FUNCTION_BLOCK FINAL FB_PackML
VAR_IN_OUT
	PackML							: ST_PMLData;
	Control							: ST_System;
END_VAR
VAR
	_Cfg_ModeTransitions			: ARRAY[0..9, 0..31] OF BOOL;
	_Index							: INT;
	_LastState						: DINT;
	_LastUnit						: DINT;
	_MessageClearPointer			: INT;
	_WarningRefreshPointer			: INT;
	_WarningRefresh					: F_TRIG;
END_VAR
VAR CONSTANT
	_MaxModeLength					: INT := 7;
	_MaxStateLength					: INT := 17;
END_VAR
VAR PERSISTENT
	_LS_H_IndicatorMatrix				: ARRAY[0..31] OF DINT :=[1032,33792,1032,361504,66784,361504,198690,67616,1028,1028,1032,99360,1216,82984,295936,1032,1028];
	_PB_IndicatorMatrix					: ARRAY[0..31] OF DINT :=[0,256,32768,0,32768,32768,32768,16384,0,256,0,0,32768,32768,16384,32768,256,0];			
	_LS_H_IndicatorDescription			: ARRAY[0..31] OF STRING(40) := ['','Alarm','Abnormal Stop','Controlled Stop','','Alert','Starved Upstream','Blocked Downstream','','','Low Material','Material Exhausted','','','Alert','Alarm','Starting / Restarting','','','','','','','','','','','','',''];		
	_PB_IndicatorDescription			: ARRAY[0..31] OF STRING(40) := ['','','','','','','','','Ready to Reset','','','','','','Ready to Start','Running','','','','','','','','','','','','','','','',''];		
END_VAR

M_Administration();
M_Commands();
M_Indicators();
M_ModeControl();
M_SafetyBreach();
M_StateMapping();
M_StateTransitions();
M_TransitionCounts();

METHOD PRIVATE M_Administration
VAR_INPUT
END_VAR
VAR_INST
	_index					: INT;
END_VAR
IF PackML.Status.UnitModeCurrent > _maxModeLength THEN
	PackML.Control.UnitMode := 0;
	PackML.Status.UnitModeCurrent := 0;
END_IF

//Time spent in Mode
//The elapsed time the machine has spent in that mode since it entered that mode.  Array index is equal to designation of the mode.
IF PackML.Status.UnitModeChangeInProcess THEN
	PackML.Admin.ModeCurrentTime[PackML.Status.UnitModeCurrent] := 0;
END_IF
IF Control.SystemTime.SecondPulse THEN
	PackML.Admin.ModeCurrentTime[PackML.Status.UnitModeCurrent] := PackML.Admin.ModeCurrentTime[PackML.Status.UnitModeCurrent] + 1;
	IF PackML.Admin.ModeCurrentTime[PackML.Status.UnitModeCurrent] < 0 THEN
		PackML.Admin.ModeCurrentTime[PackML.Status.UnitModeCurrent] := 0;
	END_IF
	IF PackML.Admin.ResetTimerCounters THEN
		FOR _index := 0 TO _maxModeLength DO
			PackML.Admin.ModeCurrentTime[_index] := 0;
		END_FOR
	END_IF
END_IF

//Cumulative TIME In Each Mode
//The cumulative elapsed time the machine has spent in each mode since it’s timers and counters were reset.  
IF Control.SystemTime.SecondPulse THEN
	PackML.Admin.ModeCummulativeTime[PackML.Status.UnitModeCurrent] := PackML.Admin.ModeCummulativeTime[PackML.Status.UnitModeCurrent] + 1;
	IF PackML.Admin.ModeCummulativeTime[PackML.Status.UnitModeCurrent] < 0 THEN
		PackML.Admin.ModeCummulativeTime[PackML.Status.UnitModeCurrent] := 0;
	END_IF
	IF PackML.Admin.ResetTimerCounters THEN
		FOR _index := 0 TO _maxModeLength DO
			PackML.Admin.ModeCummulativeTime[_index] := 0;
		END_FOR
	END_IF
END_IF

//TIME spent in State
//The elapsed time the machine has spent in that State since it entered that State.  Array index is equal to designation of the mode.
IF PackML.Status.StateChangeInProgress THEN
	PackML.Admin.StateCurrentTime[PackML.Status.UnitModeCurrent,PackML.Status.StateCurrent] := 0;
END_IF
IF Control.SystemTime.SecondPulse THEN
	PackML.Admin.StateCurrentTime[PackML.Status.UnitModeCurrent,PackML.Status.StateCurrent] := PackML.Admin.StateCurrentTime[PackML.Status.UnitModeCurrent,PackML.Status.StateCurrent] + 1;
	IF PackML.Admin.StateCurrentTime[PackML.Status.UnitModeCurrent,PackML.Status.StateCurrent] < 0 THEN
		PackML.Admin.StateCurrentTime[PackML.Status.UnitModeCurrent,PackML.Status.StateCurrent] := 0;
	END_IF
	IF PackML.Admin.ResetTimerCounters THEN
		FOR _index := 0 TO _maxStateLength DO
			PackML.Admin.StateCurrentTime[PackML.Status.UnitModeCurrent,_index] := 0;
		END_FOR
	END_IF
END_IF

//Cumulative Time In Each Mode
//The cumulative elapsed time the machine has spent in each mode since it’s timers and counters were reset.  
IF Control.SystemTime.SecondPulse THEN
	PackML.Admin.StateCummulativeTime[PackML.Status.UnitModeCurrent,PackML.Status.StateCurrent] := PackML.Admin.StateCummulativeTime[PackML.Status.UnitModeCurrent,PackML.Status.StateCurrent] + 1;
	IF PackML.Admin.StateCummulativeTime[PackML.Status.UnitModeCurrent,PackML.Status.StateCurrent] < 0 THEN
		PackML.Admin.StateCummulativeTime[PackML.Status.UnitModeCurrent,PackML.Status.StateCurrent] := 0;
	END_IF
	IF PackML.Admin.ResetTimerCounters THEN
		FOR _index := 0 TO _maxStateLength DO
			PackML.Admin.StateCummulativeTime[PackML.Status.UnitModeCurrent,_index] := 0;
		END_FOR
	END_IF
END_IF
END_METHOD

METHOD PRIVATE M_Commands
VAR_INPUT
END_VAR
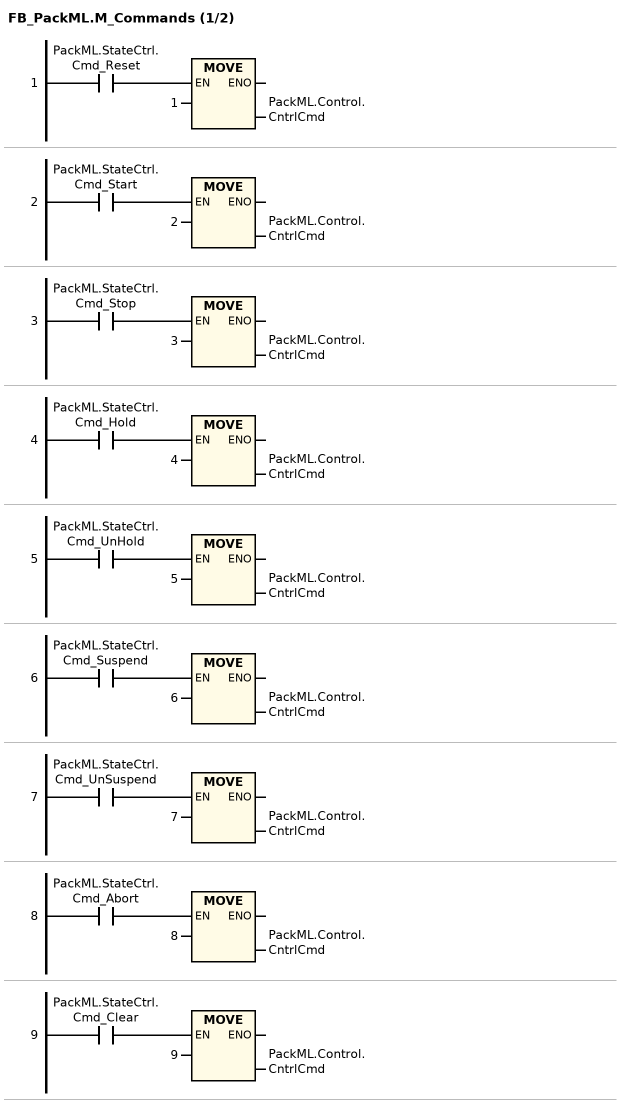
// NETWORK 1
IF PackML.StateCtrl.Cmd_Reset THEN PackML.Control.CntrlCmd := 1; END_IF

// NETWORK 2
IF PackML.StateCtrl.Cmd_Start THEN PackML.Control.CntrlCmd := 2; END_IF

// NETWORK 3
IF PackML.StateCtrl.Cmd_Stop THEN PackML.Control.CntrlCmd := 3; END_IF

// NETWORK 4
IF PackML.StateCtrl.Cmd_Hold THEN PackML.Control.CntrlCmd := 4; END_IF

// NETWORK 5
IF PackML.StateCtrl.Cmd_UnHold THEN PackML.Control.CntrlCmd := 5; END_IF

// NETWORK 6
IF PackML.StateCtrl.Cmd_Suspend THEN PackML.Control.CntrlCmd := 6; END_IF

// NETWORK 7
IF PackML.StateCtrl.Cmd_UnSuspend THEN PackML.Control.CntrlCmd := 7; END_IF

// NETWORK 8
IF PackML.StateCtrl.Cmd_Abort THEN PackML.Control.CntrlCmd := 8; END_IF

// NETWORK 9
IF PackML.StateCtrl.Cmd_Clear THEN PackML.Control.CntrlCmd := 9; END_IF

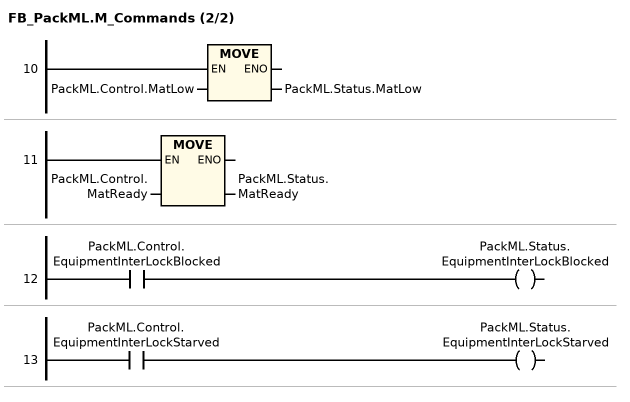
// NETWORK 10
PackML.Status.MatLow := PackML.Control.MatLow;

// NETWORK 11
PackML.Status.MatReady := PackML.Control.MatReady;

// NETWORK 12
PackML.Status.EquipmentInterLockBlocked := PackML.Control.EquipmentInterLockBlocked;

// NETWORK 13
PackML.Status.EquipmentInterLockStarved := PackML.Control.EquipmentInterLockStarved;
END_METHOD

METHOD PRIVATE M_Indicators
VAR_INST
	_i 		: DINT;
	_f_trig	: F_TRIG;
	_r_trig	: R_TRIG;
	k : bool;
END_VAR
PackML.Indicator.LS_H_Output := _LS_H_IndicatorMatrix[PackML.Status.StateCurrent];

//Red Lamp
IF PackML.Indicator.LS_H_Output.0 THEN
	PackML.Indicator.RedLamp := Control.SystemTime.PulseFlash;
ELSIF PackML.Indicator.LS_H_Output.1 AND Control.Outputs.Alarm THEN
	PackML.Indicator.RedLamp := Control.SystemTime.FastFlash;
ELSIF PackML.Indicator.LS_H_Output.2 THEN
	PackML.Indicator.RedLamp := Control.SystemTime.SlowFlash;
ELSIF PackML.Indicator.LS_H_Output.3 THEN
	PackML.Indicator.RedLamp := TRUE;
ELSE
	PackML.Indicator.RedLamp := FALSE;
END_IF

//Amber Lamp
IF PackML.Indicator.LS_H_Output.4 THEN
	PackML.Indicator.AmberLamp := Control.SystemTime.PulseFlash;
ELSIF PackML.Indicator.LS_H_Output.5 AND Control.Outputs.Alert THEN
	PackML.Indicator.AmberLamp := Control.SystemTime.FastFlash;
ELSIF PackML.Indicator.LS_H_Output.6 THEN
	PackML.Indicator.AmberLamp := Control.SystemTime.SlowFlash;
ELSIF PackML.Indicator.LS_H_Output.7 THEN
	PackML.Indicator.AmberLamp := TRUE;
ELSE
	PackML.Indicator.AmberLamp := FALSE;
END_IF

//Blue Lamp
IF PackML.Indicator.LS_H_Output.8 THEN
	PackML.Indicator.BlueLamp := Control.SystemTime.PulseFlash;
ELSIF PackML.Indicator.LS_H_Output.9 THEN
	PackML.Indicator.BlueLamp := Control.SystemTime.FastFlash;
ELSIF PackML.Indicator.LS_H_Output.10 THEN
	FOR	_i := 0 TO SIZEOF(Packml.Status.MatLow) BY 1 DO
		IF Packml.Status.MatLow[_i] THEN
			PackML.Indicator.BlueLamp := Control.SystemTime.SlowFlash;
			EXIT;
		END_IF
	END_FOR
ELSIF PackML.Indicator.LS_H_Output.11 THEN
	FOR	_i := 0 TO SIZEOF(Packml.Status.MatReady) BY 1 DO
		_f_trig(CLK:= Packml.Status.MatReady[_i]);
		IF _f_trig.Q THEN
			PackML.Indicator.BlueLamp := TRUE;
			EXIT;
		END_IF
		_r_trig(CLK:= Packml.Status.MatReady[_i]);
		IF _r_trig.Q THEN
			PackML.Indicator.BlueLamp := FALSE;
			EXIT;
		END_IF
	END_FOR
ELSE
	PackML.Indicator.BlueLamp := FALSE;
END_IF

//Green Lamp
IF PackML.Indicator.LS_H_Output.12 THEN
	PackML.Indicator.GreenLamp := Control.SystemTime.PulseFlash;
ELSIF PackML.Indicator.LS_H_Output.13 THEN
	PackML.Indicator.GreenLamp := Control.SystemTime.FastFlash;
ELSIF PackML.Indicator.LS_H_Output.14 THEN
	PackML.Indicator.GreenLamp := Control.SystemTime.SlowFlash;
ELSIF PackML.Indicator.LS_H_Output.15 THEN
	PackML.Indicator.GreenLamp := TRUE;
ELSE
	PackML.Indicator.GreenLamp := FALSE;
END_IF

//Horn
IF PackML.Indicator.LS_H_Output.16 AND Control.Outputs.Alert THEN
	PackML.Indicator.Horn := Control.SystemTime.PulseFlash;
ELSIF PackML.Indicator.LS_H_Output.17 AND Control.Outputs.Alarm THEN
	PackML.Indicator.Horn := Control.SystemTime.FastFlash;
ELSIF PackML.Indicator.LS_H_Output.18 THEN
	PackML.Indicator.Horn := Control.SystemTime.SlowFlash;
ELSIF PackML.Indicator.LS_H_Output.19 THEN
	PackML.Indicator.Horn := TRUE;
ELSE
	PackML.Indicator.Horn := FALSE;
END_IF

PackML.Indicator.PB_Output := _PB_IndicatorMatrix[PackML.Status.StateCurrent];

//Red Button
IF PackML.Indicator.PB_Output.0 THEN
	PackML.Indicator.RedButton := Control.SystemTime.PulseFlash;
ELSIF PackML.Indicator.PB_Output.1 THEN
	PackML.Indicator.RedButton := Control.SystemTime.FastFlash;
ELSIF PackML.Indicator.PB_Output.2 THEN
	PackML.Indicator.RedButton := Control.SystemTime.SlowFlash;
ELSIF PackML.Indicator.PB_Output.3 THEN
	PackML.Indicator.RedButton := TRUE;
ELSE
	PackML.Indicator.RedButton := FALSE;
END_IF

//Amber Button
IF PackML.Indicator.PB_Output.4 THEN
	PackML.Indicator.AmberButton := Control.SystemTime.PulseFlash;
ELSIF PackML.Indicator.PB_Output.5 THEN
	PackML.Indicator.AmberButton := Control.SystemTime.FastFlash;
ELSIF PackML.Indicator.PB_Output.6 THEN
	PackML.Indicator.AmberButton := Control.SystemTime.SlowFlash;
ELSIF PackML.Indicator.PB_Output.7 THEN
	PackML.Indicator.AmberButton := TRUE;
ELSE
	PackML.Indicator.AmberButton := FALSE;
END_IF

//Blue Button
IF PackML.Indicator.PB_Output.8 THEN
	PackML.Indicator.BlueButton := Control.SystemTime.PulseFlash;
ELSIF PackML.Indicator.PB_Output.9 THEN
	PackML.Indicator.BlueButton := Control.SystemTime.FastFlash;
ELSIF PackML.Indicator.PB_Output.10 THEN
	PackML.Indicator.BlueButton := Control.SystemTime.SlowFlash;
ELSIF PackML.Indicator.PB_Output.11 THEN
	PackML.Indicator.BlueButton := TRUE;
ELSE
	PackML.Indicator.BlueButton := FALSE;
END_IF

//Green Button
IF PackML.Indicator.PB_Output.12 THEN
	PackML.Indicator.GreenButton := Control.SystemTime.PulseFlash;
ELSIF PackML.Indicator.PB_Output.13 THEN
	PackML.Indicator.GreenButton := Control.SystemTime.FastFlash;
ELSIF PackML.Indicator.PB_Output.14 THEN
	PackML.Indicator.GreenButton := Control.SystemTime.SlowFlash;
ELSIF PackML.Indicator.PB_Output.15 THEN
	PackML.Indicator.GreenButton := TRUE;
ELSE
	PackML.Indicator.GreenButton := FALSE;
END_IF
END_METHOD

METHOD PRIVATE M_ModeControl
VAR_INPUT
END_VAR
VAR_INST
END_VAR
IF Control.SystemTime.FirstCycle THEN
	FOR _index := 0 TO 9 BY 1 DO
		_cfg_ModeTransitions[_index,2] := TRUE;
		_cfg_ModeTransitions[_index,9] := TRUE;
	END_FOR
END_IF

IF PackML.Control.UnitMode >= 1 AND PackML.Control.UnitMode <= 32 AND (PackML.Control.UnitMode <> PackML.Status.UnitModeCurrent) THEN
	IF _cfg_ModeTransitions[PackML.Status.UnitModeCurrent,PackML.Status.StateCurrent] AND _cfg_ModeTransitions[PackML.Control.UnitMode,PackML.Status.StateCurrent] THEN
		PackML.Status.UnitModeCurrent := PackML.Control.UnitMode;
	END_IF
	PackML.Control.UnitModeChangeRequest := TRUE;
	PackML.Status.UnitModeRequested := TRUE;
ELSE
	PackML.Control.UnitModeChangeRequest := FALSE;
	PackML.Status.UnitModeRequested := FALSE;
END_IF
END_METHOD

METHOD PRIVATE M_SafetyBreach
VAR_INPUT
END_VAR
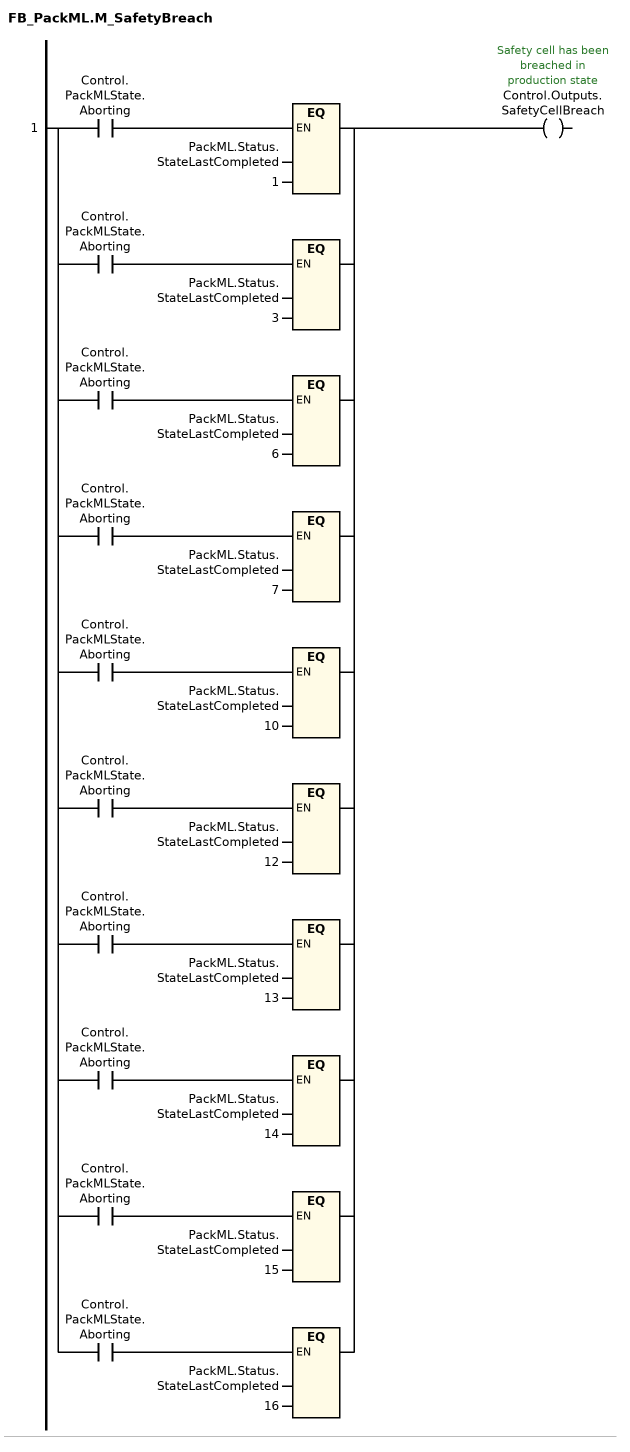
// NETWORK 1
//   PackML.Status.StateLastCompleted: Last Completed State
//   Control.Outputs.SafetyCellBreach: Safety cell has been breached in production state
Control.Outputs.SafetyCellBreach := Control.PackMLState.Aborting AND PackML.Status.StateLastCompleted = 1 OR Control.PackMLState.Aborting AND PackML.Status.StateLastCompleted = 3 OR Control.PackMLState.Aborting AND PackML.Status.StateLastCompleted = 6 OR Control.PackMLState.Aborting AND PackML.Status.StateLastCompleted = 7 OR Control.PackMLState.Aborting AND PackML.Status.StateLastCompleted = 10 OR Control.PackMLState.Aborting AND PackML.Status.StateLastCompleted = 12 OR Control.PackMLState.Aborting AND PackML.Status.StateLastCompleted = 13 OR Control.PackMLState.Aborting AND PackML.Status.StateLastCompleted = 14 OR Control.PackMLState.Aborting AND PackML.Status.StateLastCompleted = 15 OR Control.PackMLState.Aborting AND PackML.Status.StateLastCompleted = 16;
END_METHOD

METHOD PRIVATE M_StateMapping
VAR_INPUT
END_VAR
VAR_INST
END_VAR
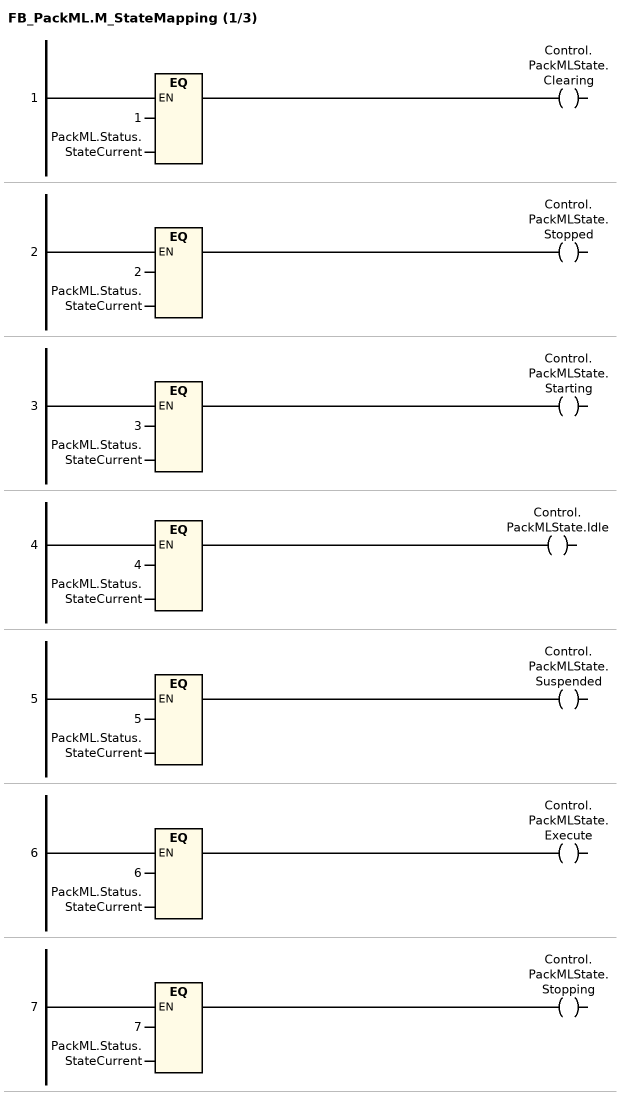
// NETWORK 1
//   PackML.Status.StateCurrent: Current State Number
Control.PackMLState.Clearing := 1 = PackML.Status.StateCurrent;

// NETWORK 2
//   PackML.Status.StateCurrent: Current State Number
Control.PackMLState.Stopped := 2 = PackML.Status.StateCurrent;

// NETWORK 3
//   PackML.Status.StateCurrent: Current State Number
Control.PackMLState.Starting := 3 = PackML.Status.StateCurrent;

// NETWORK 4
//   PackML.Status.StateCurrent: Current State Number
Control.PackMLState.Idle := 4 = PackML.Status.StateCurrent;

// NETWORK 5
//   PackML.Status.StateCurrent: Current State Number
Control.PackMLState.Suspended := 5 = PackML.Status.StateCurrent;

// NETWORK 6
//   PackML.Status.StateCurrent: Current State Number
Control.PackMLState.Execute := 6 = PackML.Status.StateCurrent;

// NETWORK 7
//   PackML.Status.StateCurrent: Current State Number
Control.PackMLState.Stopping := 7 = PackML.Status.StateCurrent;

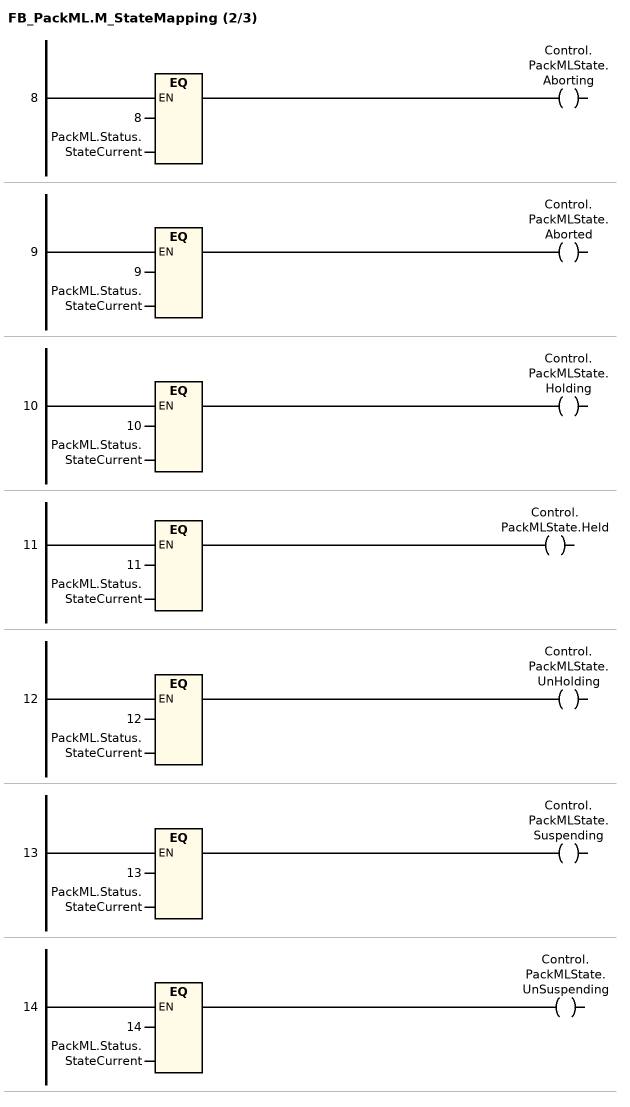
// NETWORK 8
//   PackML.Status.StateCurrent: Current State Number
Control.PackMLState.Aborting := 8 = PackML.Status.StateCurrent;

// NETWORK 9
//   PackML.Status.StateCurrent: Current State Number
Control.PackMLState.Aborted := 9 = PackML.Status.StateCurrent;

// NETWORK 10
//   PackML.Status.StateCurrent: Current State Number
Control.PackMLState.Holding := 10 = PackML.Status.StateCurrent;

// NETWORK 11
//   PackML.Status.StateCurrent: Current State Number
Control.PackMLState.Held := 11 = PackML.Status.StateCurrent;

// NETWORK 12
//   PackML.Status.StateCurrent: Current State Number
Control.PackMLState.UnHolding := 12 = PackML.Status.StateCurrent;

// NETWORK 13
//   PackML.Status.StateCurrent: Current State Number
Control.PackMLState.Suspending := 13 = PackML.Status.StateCurrent;

// NETWORK 14
//   PackML.Status.StateCurrent: Current State Number
Control.PackMLState.UnSuspending := 14 = PackML.Status.StateCurrent;

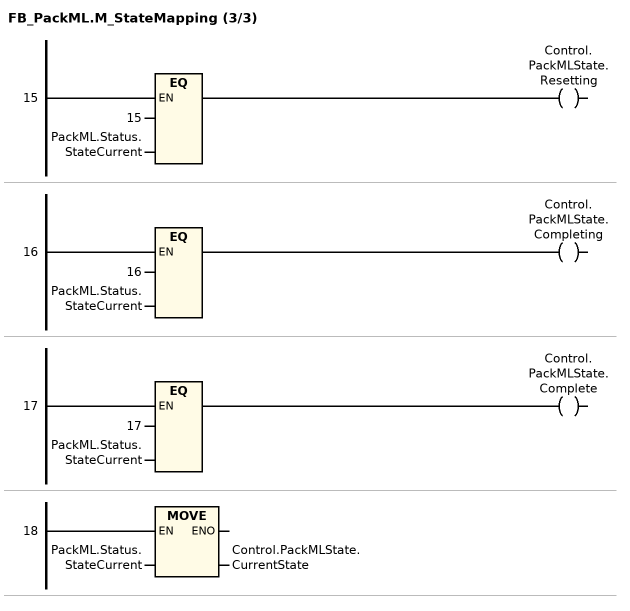
// NETWORK 15
//   PackML.Status.StateCurrent: Current State Number
Control.PackMLState.Resetting := 15 = PackML.Status.StateCurrent;

// NETWORK 16
//   PackML.Status.StateCurrent: Current State Number
Control.PackMLState.Completing := 16 = PackML.Status.StateCurrent;

// NETWORK 17
//   PackML.Status.StateCurrent: Current State Number
Control.PackMLState.Complete := 17 = PackML.Status.StateCurrent;

// NETWORK 18
//   PackML.Status.StateCurrent: Current State Number
Control.PackMLState.CurrentState := PackML.Status.StateCurrent;
END_METHOD

METHOD PRIVATE M_StateTransitions
VAR_INPUT
END_VAR
VAR_INST
END_VAR
//Clearing - 1
IF Control.PackMLState.Aborted AND PackML.StateCtrl.Cmd_Clear THEN
	PackML.Control.State := 1;
	PackML.Status.StateLastCompleted := PackML.Status.StateCurrent;
	PackML.Status.StateCurrent := PackML.Control.State;
END_IF

//Stopped - 2
IF Control.PackMLState.Stopping OR Control.PackMLState.Clearing THEN
	PackML.Control.State := 2;
	IF PackML.Control.StateChangeRequest THEN
		PackML.Status.StateLastCompleted := PackML.Status.StateCurrent;
		PackML.Status.StateCurrent := PackML.Control.State;
	END_IF
END_IF

//Starting - 3
IF Control.PackMLState.Idle AND PackML.StateCtrl.Cmd_Start THEN
	PackML.Control.State := 3;
	PackML.Status.StateLastCompleted := PackML.Status.StateCurrent;
	PackML.Status.StateCurrent := PackML.Control.State;
END_IF

//Idle - 4
IF Control.PackMLState.Resetting THEN
	PackML.Control.State := 4;
	IF PackML.Control.StateChangeRequest THEN
		PackML.Status.StateLastCompleted := PackML.Status.StateCurrent;
		PackML.Status.StateCurrent := PackML.Control.State;
	END_IF
END_IF

//Suspended - 5
IF Control.PackMLState.Suspending THEN
	PackML.Control.State := 5;
	IF PackML.Control.StateChangeRequest THEN
		PackML.Status.StateLastCompleted := PackML.Status.StateCurrent;
		PackML.Status.StateCurrent := PackML.Control.State;
	END_IF
END_IF

//Execute - 6
IF Control.PackMLState.Starting OR Control.PackMLState.UnHolding OR Control.PackMLState.UnSuspending THEN
	PackML.Control.State := 6;
	IF PackML.Control.StateChangeRequest THEN
		PackML.Status.StateLastCompleted := PackML.Status.StateCurrent;
		PackML.Status.StateCurrent := PackML.Control.State;
	END_IF
END_IF

//Stopping - 7
IF (Control.PackMLState.Resetting 
OR Control.PackMLState.Idle 
OR Control.PackMLState.Starting 
OR Control.PackMLState.Execute 
OR Control.PackMLState.Holding 
OR Control.PackMLState.Held 
OR Control.PackMLState.UnHolding 
OR Control.PackMLState.Suspending
OR Control.PackMLState.Suspended
OR Control.PackMLState.UnSuspending 
OR Control.PackMLState.Completing 
OR Control.PackMLState.Clearing 
OR Control.PackMLState.Complete) 
AND PackML.StateCtrl.Cmd_Stop THEN
	PackML.Control.State := 7;
	PackML.Status.StateLastCompleted := PackML.Status.StateCurrent;
	PackML.Status.StateCurrent := PackML.Control.State;
END_IF

//Aborting - 8
IF (NOT Control.PackMLState.Aborting AND NOT Control.PackMLState.Aborted AND PackML.StateCtrl.Cmd_Abort) 
OR (PackML.Control.State <= 0 OR PackML.Control.State >= 18) 
OR (PackML.Status.StateCurrent <= 0 OR PackML.Status.StateCurrent >= 18)  THEN
	PackML.Control.State := 8;
	PackML.Status.StateLastCompleted := PackML.Status.StateCurrent;
	PackML.Status.StateCurrent := PackML.Control.State;
END_IF

//Abort - 9
IF Control.PackMLState.Aborting THEN
	PackML.Control.State := 9;
	IF PackML.Control.StateChangeRequest THEN
		PackML.Status.StateLastCompleted := PackML.Status.StateCurrent;
		PackML.Status.StateCurrent := PackML.Control.State;
	END_IF
END_IF

//Holding - 10
IF Control.PackMLState.Execute AND PackML.StateCtrl.Cmd_Hold THEN
	PackML.Control.State := 10;
	PackML.Status.StateLastCompleted := PackML.Status.StateCurrent;
	PackML.Status.StateCurrent := PackML.Control.State;
END_IF

//Held - 11
IF Control.PackMLState.Holding THEN
	PackML.Control.State := 11;
	IF PackML.Control.StateChangeRequest THEN
		PackML.Status.StateLastCompleted := PackML.Status.StateCurrent;
		PackML.Status.StateCurrent := PackML.Control.State;
	END_IF
END_IF

//Unholding - 12
IF Control.PackMLState.Held AND PackML.StateCtrl.Cmd_UnHold THEN
	PackML.Control.State := 12;
	PackML.Status.StateLastCompleted := PackML.Status.StateCurrent;
	PackML.Status.StateCurrent := PackML.Control.State;
END_IF

//Suspending - 13
IF Control.PackMLState.Execute AND PackML.StateCtrl.Cmd_Suspend THEN
	PackML.Control.State := 13;
	PackML.Status.StateLastCompleted := PackML.Status.StateCurrent;
	PackML.Status.StateCurrent := PackML.Control.State;
END_IF

//UnSuspending - 14
IF Control.PackMLState.Suspended AND PackML.StateCtrl.Cmd_UnSuspend THEN
	PackML.Control.State := 14;
	PackML.Status.StateLastCompleted := PackML.Status.StateCurrent;
	PackML.Status.StateCurrent := PackML.Control.State;
END_IF

//Resetting - 15
IF (Control.PackMLState.Stopped 
OR Control.PackMLState.Complete)
AND PackML.StateCtrl.Cmd_Reset THEN
	PackML.Control.State := 15;
	PackML.Status.StateLastCompleted := PackML.Status.StateCurrent;
	PackML.Status.StateCurrent := PackML.Control.State;
END_IF

//Completing - 16
IF Control.PackMLState.Execute AND PackML.StateCtrl.Sts_Execute_SC THEN
	PackML.Control.State := 16;
	PackML.Status.StateLastCompleted := PackML.Status.StateCurrent;
	PackML.Status.StateCurrent := PackML.Control.State;
END_IF

//Complete - 17
IF Control.PackMLState.Completing THEN
	PackML.Control.State := 17;
	IF PackML.Control.StateChangeRequest THEN
		PackML.Status.StateLastCompleted := PackML.Status.StateCurrent;
		PackML.Status.StateCurrent := PackML.Control.State;
	END_IF
END_IF
END_METHOD

METHOD PRIVATE M_TransitionCounts
VAR_INPUT
END_VAR
VAR_INST
END_VAR
VAR_INST // added by the converter: edge detectors and wires of the graphical bodies
    _w1, _w2 : BOOL;
END_VAR
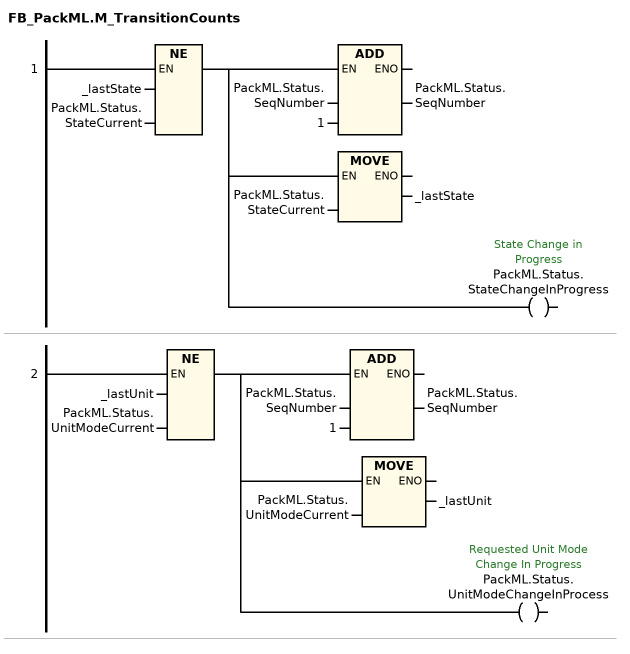
// NETWORK 1
//   PackML.Status.StateCurrent: Current State Number
//   PackML.Status.SeqNumber: Pack ML Sequence Number
//   PackML.Status.StateChangeInProgress: State Change in Progress
_w1 := _lastState <> PackML.Status.StateCurrent;
IF _w1 THEN PackML.Status.SeqNumber := PackML.Status.SeqNumber + 1; END_IF
IF _w1 THEN _lastState := PackML.Status.StateCurrent; END_IF
PackML.Status.StateChangeInProgress := _w1;

// NETWORK 2
//   PackML.Status.UnitModeCurrent: Unit Mode in current use
//   PackML.Status.SeqNumber: Pack ML Sequence Number
//   PackML.Status.UnitModeChangeInProcess: Requested Unit Mode Change In Progress
_w2 := _lastUnit <> PackML.Status.UnitModeCurrent;
IF _w2 THEN PackML.Status.SeqNumber := PackML.Status.SeqNumber + 1; END_IF
IF _w2 THEN _lastUnit := PackML.Status.UnitModeCurrent; END_IF
PackML.Status.UnitModeChangeInProcess := _w2;
END_METHOD

END_FUNCTION_BLOCK

(* stored: Version 1.1.0.1, ProductVersion 3.1.4024.3
   POU FB_PackML: Id {dd9d0941-a275-4cce-82d7-a4caaca448cb}, SpecialFunc None
   Method M_Administration: Id {57d57029-ae39-4d00-bcb2-216a553f7f2f}
   Method M_Commands: Id {a1bf88f9-d37a-43f4-b2b2-9b73c6351052}
   Method M_Indicators: Id {5a6cfd73-1311-457f-b58b-c422e87453d9}
   Method M_ModeControl: Id {896a59e0-7969-4c92-960b-48e14562a8b8}
   Method M_SafetyBreach: Id {d6c0d60e-06b5-49d9-8849-985f77d46e8f}
   Method M_StateMapping: Id {df009cd7-0641-44da-9ace-57ee4b47ee8b}
   Method M_StateTransitions: Id {fdecf6b2-9f49-492d-9e0c-11b673d5a5b5}
   Method M_TransitionCounts: Id {19bb2792-b1a2-4685-900f-3fa206734dbd} *)
